PROGRAM MAIN
VAR

END_VAR

POU_readSupvData();
POU_writeReactorToSupvData();

END_PROGRAM

(* stored: Version 1.1.0.1, ProductVersion 3.1.4024.11
   POU MAIN: Id {5d841a3c-4032-4429-ae88-cfe024ef2812}, SpecialFunc None *)
